(* PLC project  *)

CONFIGURATION phyBOARD_Lyra
END_CONFIGURATION
